PROGRAM MAIN
VAR
END_VAR

ModelExecution();

END_PROGRAM

(* stored: Version 1.1.0.1, ProductVersion 3.1.4024.4
   POU MAIN: Id {2969ad3f-3f42-48b3-843e-ab7901aced5d}, SpecialFunc None *)
